FUNCTION_BLOCK SP_ExtendPlunger (* ExtendPlunger parameters (Duration [s] 0.0..20.0, default 10.0): OPC UA IDs, range check and latching *)
  (* Standard: 61499-2 *)
  (* Version 0.1, 2026-09-28, Project contributors, AAU Smart Production Lab *)
  PACKAGE stoppering;
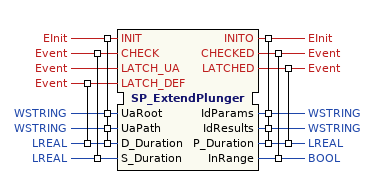
  EVENT_INPUT
    INIT : EInit WITH UaRoot, UaPath, D_Duration;
    CHECK WITH S_Duration;
    LATCH_UA;
    LATCH_DEF WITH D_Duration;
  END_EVENT
  EVENT_OUTPUT
    INITO : EInit WITH IdParams, IdResults, P_Duration;
    CHECKED WITH InRange;
    LATCHED WITH P_Duration;
  END_EVENT
  VAR_INPUT
    UaRoot : WSTRING;
    UaPath : WSTRING;
    D_Duration : LREAL;
    S_Duration : LREAL;
  END_VAR
  VAR_OUTPUT
    IdParams : WSTRING;
    IdResults : WSTRING;
    P_Duration : LREAL;
    InRange : BOOL;
  END_VAR
  EC_STATES
    INIT : INIT -> INITO;
    CHECK : CHECK -> CHECKED;
    LATCH_UA : LATCH_UA -> LATCHED;
    LATCH_DEF : LATCH_DEF -> LATCHED;
  END_STATES
  ALGORITHM INIT IN ST:
IdParams := CONCAT(CONCAT(CONCAT("opc_ua[WRITE;", CONCAT(UaRoot, UaPath)), "/Parameters/Duration"), "]");
IdResults := "";
P_Duration := D_Duration;
  END_ALGORITHM
  ALGORITHM CHECK IN ST:
InRange := (S_Duration >= 0.0) AND (S_Duration <= 20.0);
  END_ALGORITHM
  ALGORITHM LATCH_UA IN ST:
P_Duration := S_Duration;
  END_ALGORITHM
  ALGORITHM LATCH_DEF IN ST:
P_Duration := D_Duration;
  END_ALGORITHM
END_FUNCTION_BLOCK
